# EPICS substitutions: RadiationMonitoringApp/Db/sioc-bsyh-rm01.substitutions
file radm_info.template {
    pattern
    {             P,       LOC, TYPE }
    { RADM:BSYH:843, "BSYH D2",    0 }
}

file fhtCommon.template {
    pattern
    {             P,         PORT }
    { RADM:BSYH:843, FHT_BSYH_843 }
}

file fhtChan.template {
    pattern
    {             P,         PORT,  N,  M }
    { RADM:BSYH:843, FHT_BSYH_843, 01,  1 }
    { RADM:BSYH:843, FHT_BSYH_843, 02,  2 }
    { RADM:BSYH:843, FHT_BSYH_843, 03,  3 }
    { RADM:BSYH:843, FHT_BSYH_843, 04,  4 }
    { RADM:BSYH:843, FHT_BSYH_843, 05,  5 }
    { RADM:BSYH:843, FHT_BSYH_843, 06,  6 }
    { RADM:BSYH:843, FHT_BSYH_843, 07,  7 }
    { RADM:BSYH:843, FHT_BSYH_843, 08,  8 }
    { RADM:BSYH:843, FHT_BSYH_843, 09,  9 }
    { RADM:BSYH:843, FHT_BSYH_843, 10, 10 }
    { RADM:BSYH:843, FHT_BSYH_843, 11, 11 }
    { RADM:BSYH:843, FHT_BSYH_843, 12, 12 }
    { RADM:BSYH:843, FHT_BSYH_843, 13, 13 }
    { RADM:BSYH:843, FHT_BSYH_843, 14, 14 }
    { RADM:BSYH:843, FHT_BSYH_843, 15, 15 }
    { RADM:BSYH:843, FHT_BSYH_843, 16, 16 }
}

file fht40G.template {
    pattern
    {             P,         PORT,  N,  M }
    { RADM:BSYH:843, FHT_BSYH_843, 01,  1 }
    { RADM:BSYH:843, FHT_BSYH_843, 02,  2 }
}

file fhtChanDisplay.template {
    pattern
    {             P,         PORT,  N }
    { RADM:BSYH:843, FHT_BSYH_843, 01 }
    { RADM:BSYH:843, FHT_BSYH_843, 02 }
    { RADM:BSYH:843, FHT_BSYH_843, 03 }
}
